// TIA Portal V15.1 export
// export: Created 2024-05-17T05:38:59.4838235Z, ExportSetting WithDefaults, DisplayName Totally Integrated Automation Portal, DisplayVersion V15.1 Update 5, DisplayName TIA Portal Openness, DisplayVersion V15.1 Update 5, DisplayName SINAMICS Startdrive Advanced, DisplayVersion V15.1, DisplayName G130, G150, S120, S150, SINAMICS MV, S210, DisplayVersion V15.1, DisplayName G110M, G120, G120C, G120D, G120P, DisplayVersion V15.1, DisplayName STEP 7 Professional, DisplayVersion V15.1 Update 5, DisplayName STEP 7 Safety, DisplayVersion V15.1, DisplayName WinCC Professional, DisplayVersion V15.1 Update 5, DisplayName SIMATIC Visualization Architect, DisplayVersion V15.1
FUNCTION "DiagPLCOverview" : Void   // FC251, FBD
TITLE = DiagPLCOverview
{ S7_Optimized_Access := 'FALSE' }
AUTHOR : VCC
NAME : LocFunc
VERSION : 0.1
// stored: AutoNumber false, IsIECCheckEnabled false, SetENOAutomatically False, UDAEnableTagReadback false
   VAR_OUTPUT
      O_AlarmA : Bool;   // Alarm A
      O_AlarmB : Bool;   // Alarm B
      O_AlarmC : Bool;   // Alarm C
      O_AlarmD : Bool;   // Alarm D
      O_AlarmABCondition : Bool;   // Alarms resetable
      H_IAnim : Word;   // Icon Animation
   END_VAR
   VAR_TEMP   // added for the SCL form of the ladder/FBD networks
      _w1 : Bool;
      _w2 : Bool;
   END_VAR
BEGIN

REGION Network 1: **** 1 - Inputs **** HMI Cmd
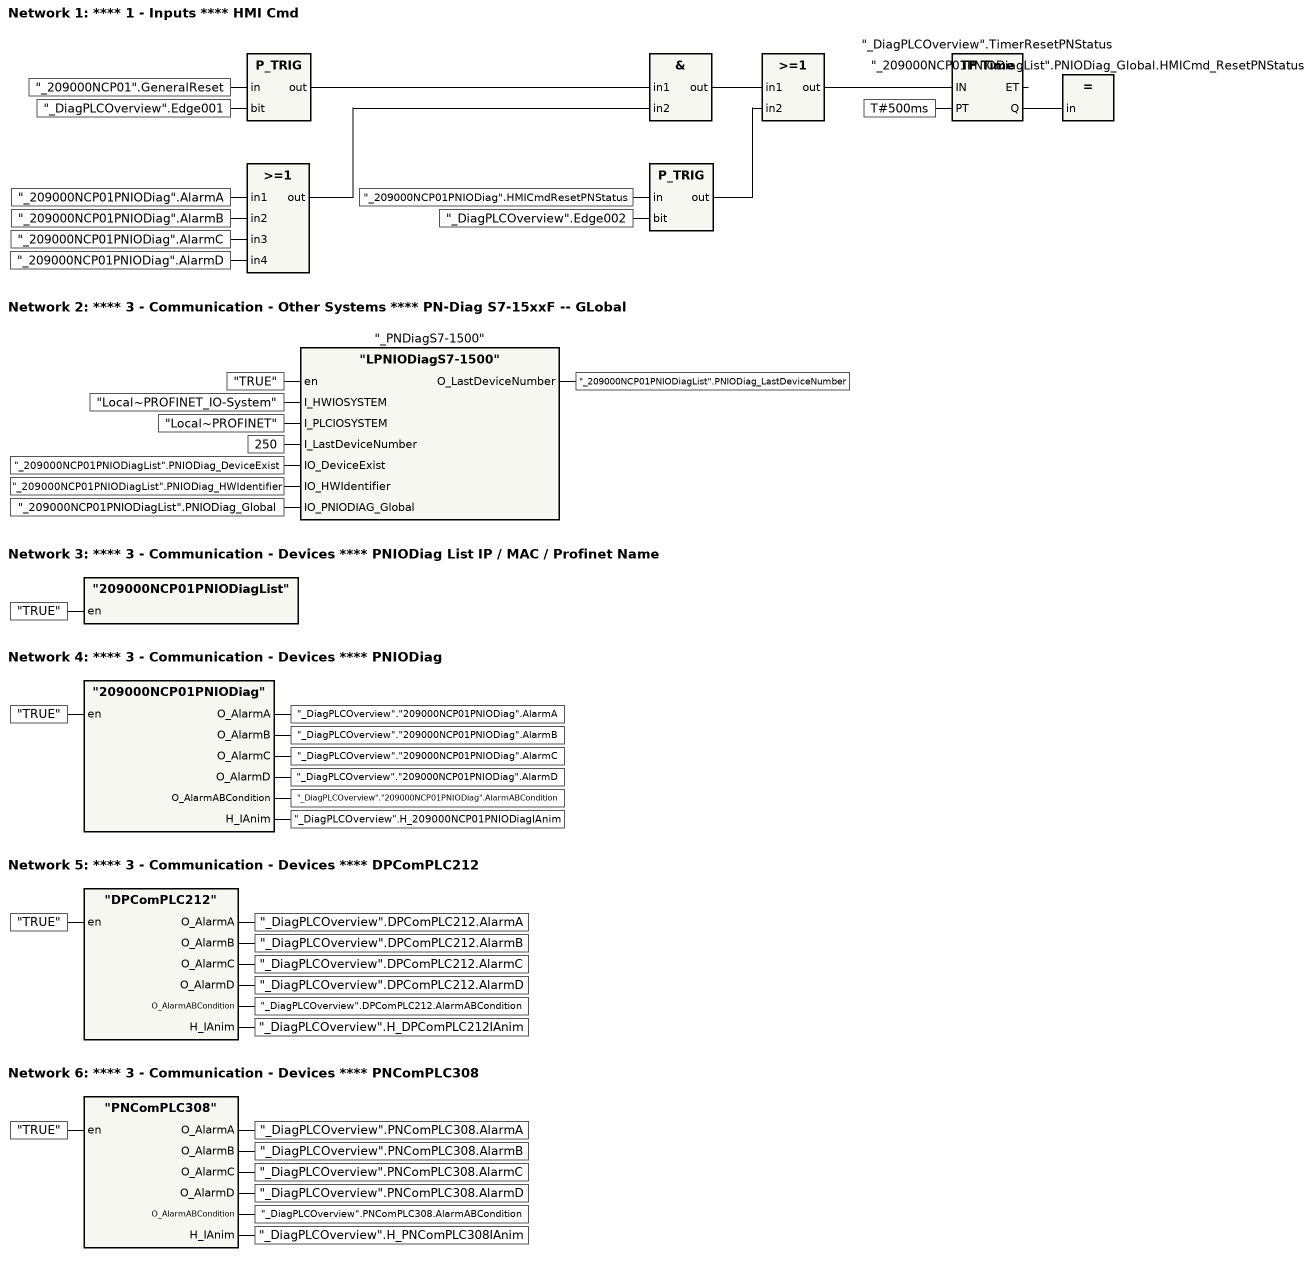
   #_w1 := "_209000NCP01".GeneralReset AND NOT "_DiagPLCOverview".Edge001;   // rising edge
   "_DiagPLCOverview".Edge001 := "_209000NCP01".GeneralReset;
   #_w2 := "_209000NCP01PNIODiag".HMICmdResetPNStatus AND NOT "_DiagPLCOverview".Edge002;   // rising edge
   "_DiagPLCOverview".Edge002 := "_209000NCP01PNIODiag".HMICmdResetPNStatus;
   "_DiagPLCOverview".TimerResetPNStatus.TP(IN := (#_w1 AND ("_209000NCP01PNIODiag".AlarmA OR "_209000NCP01PNIODiag".AlarmB OR "_209000NCP01PNIODiag".AlarmC OR "_209000NCP01PNIODiag".AlarmD)) OR #_w2,
                           PT := T#500ms);
   "_209000NCP01PNIODiagList".PNIODiag_Global.HMICmd_ResetPNStatus := "_DiagPLCOverview".TimerResetPNStatus.Q;
END_REGION

REGION Network 2: **** 3 - Communication - Other Systems **** PN-Diag S7-15xxF -- GLobal
   // PN-Diag S7-15xxF
   IF "TRUE" THEN
       "_PNDiagS7-1500"(I_HWIOSYSTEM := "Local~PROFINET_IO-System",   // "LPNIODiagS7-1500"
                        I_PLCIOSYSTEM := "Local~PROFINET",
                        I_LastDeviceNumber := 250,
                        IO_DeviceExist := "_209000NCP01PNIODiagList".PNIODiag_DeviceExist,
                        IO_HWIdentifier := "_209000NCP01PNIODiagList".PNIODiag_HWIdentifier,
                        IO_PNIODIAG_Global := "_209000NCP01PNIODiagList".PNIODiag_Global,
                        O_LastDeviceNumber => "_209000NCP01PNIODiagList".PNIODiag_LastDeviceNumber);
   END_IF;
END_REGION

REGION Network 3: **** 3 - Communication - Devices **** PNIODiag List IP / MAC / Profinet Name
   IF "TRUE" THEN "209000NCP01PNIODiagList"(); END_IF;
END_REGION

REGION Network 4: **** 3 - Communication - Devices **** PNIODiag
   IF "TRUE" THEN
       "209000NCP01PNIODiag"(O_AlarmA => "_DiagPLCOverview"."209000NCP01PNIODiag".AlarmA,
                             O_AlarmB => "_DiagPLCOverview"."209000NCP01PNIODiag".AlarmB,
                             O_AlarmC => "_DiagPLCOverview"."209000NCP01PNIODiag".AlarmC,
                             O_AlarmD => "_DiagPLCOverview"."209000NCP01PNIODiag".AlarmD,
                             O_AlarmABCondition => "_DiagPLCOverview"."209000NCP01PNIODiag".AlarmABCondition,
                             H_IAnim => "_DiagPLCOverview".H_209000NCP01PNIODiagIAnim);
   END_IF;
END_REGION

REGION Network 5: **** 3 - Communication - Devices **** DPComPLC212
   // DP/DP coupler communication
   IF "TRUE" THEN
       "DPComPLC212"(O_AlarmA => "_DiagPLCOverview".DPComPLC212.AlarmA,
                     O_AlarmB => "_DiagPLCOverview".DPComPLC212.AlarmB,
                     O_AlarmC => "_DiagPLCOverview".DPComPLC212.AlarmC,
                     O_AlarmD => "_DiagPLCOverview".DPComPLC212.AlarmD,
                     O_AlarmABCondition => "_DiagPLCOverview".DPComPLC212.AlarmABCondition,
                     H_IAnim => "_DiagPLCOverview".H_DPComPLC212IAnim);
   END_IF;
END_REGION

REGION Network 6: **** 3 - Communication - Devices **** PNComPLC308
   // PN/PN coupler communication
   IF "TRUE" THEN
       "PNComPLC308"(O_AlarmA => "_DiagPLCOverview".PNComPLC308.AlarmA,
                     O_AlarmB => "_DiagPLCOverview".PNComPLC308.AlarmB,
                     O_AlarmC => "_DiagPLCOverview".PNComPLC308.AlarmC,
                     O_AlarmD => "_DiagPLCOverview".PNComPLC308.AlarmD,
                     O_AlarmABCondition => "_DiagPLCOverview".PNComPLC308.AlarmABCondition,
                     H_IAnim => "_DiagPLCOverview".H_PNComPLC308IAnim);
   END_IF;
END_REGION

REGION Network 7: **** 3 - Communication - Devices **** VD Com
   // Virtual Device communication
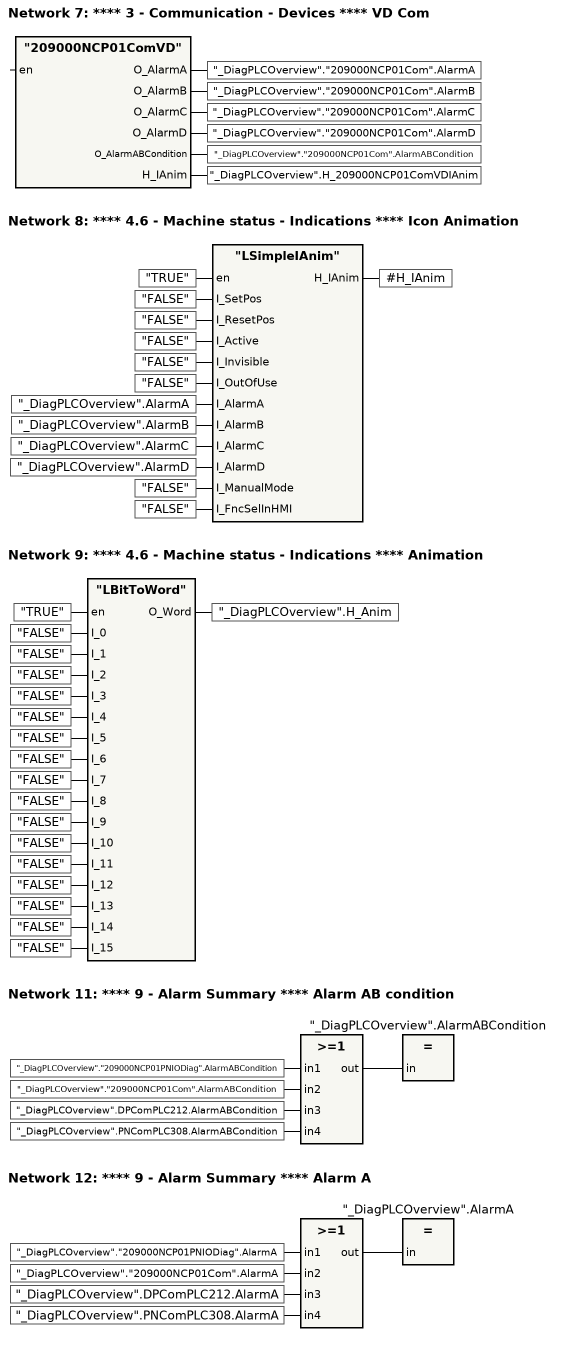
   "209000NCP01ComVD"(O_AlarmA => "_DiagPLCOverview"."209000NCP01Com".AlarmA,
                      O_AlarmB => "_DiagPLCOverview"."209000NCP01Com".AlarmB,
                      O_AlarmC => "_DiagPLCOverview"."209000NCP01Com".AlarmC,
                      O_AlarmD => "_DiagPLCOverview"."209000NCP01Com".AlarmD,
                      O_AlarmABCondition => "_DiagPLCOverview"."209000NCP01Com".AlarmABCondition,
                      H_IAnim => "_DiagPLCOverview".H_209000NCP01ComVDIAnim);
END_REGION

REGION Network 8: **** 4.6 - Machine status - Indications **** Icon Animation
   // Icon Animation for HMI
   IF "TRUE" THEN
       "LSimpleIAnim"(I_SetPos := "FALSE",
                      I_ResetPos := "FALSE",
                      I_Active := "FALSE",
                      I_Invisible := "FALSE",
                      I_OutOfUse := "FALSE",
                      I_AlarmA := "_DiagPLCOverview".AlarmA,
                      I_AlarmB := "_DiagPLCOverview".AlarmB,
                      I_AlarmC := "_DiagPLCOverview".AlarmC,
                      I_AlarmD := "_DiagPLCOverview".AlarmD,
                      I_ManualMode := "FALSE",
                      I_FncSelInHMI := "FALSE",
                      H_IAnim => #H_IAnim);
   END_IF;
END_REGION

REGION Network 9: **** 4.6 - Machine status - Indications **** Animation
   // Animation
   IF "TRUE" THEN
       "LBitToWord"(I_0 := "FALSE",
                    I_1 := "FALSE",
                    I_2 := "FALSE",
                    I_3 := "FALSE",
                    I_4 := "FALSE",
                    I_5 := "FALSE",
                    I_6 := "FALSE",
                    I_7 := "FALSE",
                    I_8 := "FALSE",
                    I_9 := "FALSE",
                    I_10 := "FALSE",
                    I_11 := "FALSE",
                    I_12 := "FALSE",
                    I_13 := "FALSE",
                    I_14 := "FALSE",
                    I_15 := "FALSE",
                    O_Word => "_DiagPLCOverview".H_Anim);
   END_IF;
END_REGION

NETWORK
TITLE = **** 4.6 - Machine Status - Indications **** Animation DB number
// DB number
      OPN   "_DiagPLCOverview";
      L     DBNO;
      T     "_DiagPLCOverview".H_DBnr;

REGION Network 11: **** 9 - Alarm Summary **** Alarm AB condition
   // Alarm AB condition
   "_DiagPLCOverview".AlarmABCondition := "_DiagPLCOverview"."209000NCP01PNIODiag".AlarmABCondition OR "_DiagPLCOverview"."209000NCP01Com".AlarmABCondition OR "_DiagPLCOverview".DPComPLC212.AlarmABCondition OR "_DiagPLCOverview".PNComPLC308.AlarmABCondition;
END_REGION

REGION Network 12: **** 9 - Alarm Summary **** Alarm A
   // Summary of alarms A
   "_DiagPLCOverview".AlarmA := "_DiagPLCOverview"."209000NCP01PNIODiag".AlarmA OR "_DiagPLCOverview"."209000NCP01Com".AlarmA OR "_DiagPLCOverview".DPComPLC212.AlarmA OR "_DiagPLCOverview".PNComPLC308.AlarmA;
END_REGION

REGION Network 13: **** 9 - Alarm Summary **** Alarm B
   // Summary of alarms B
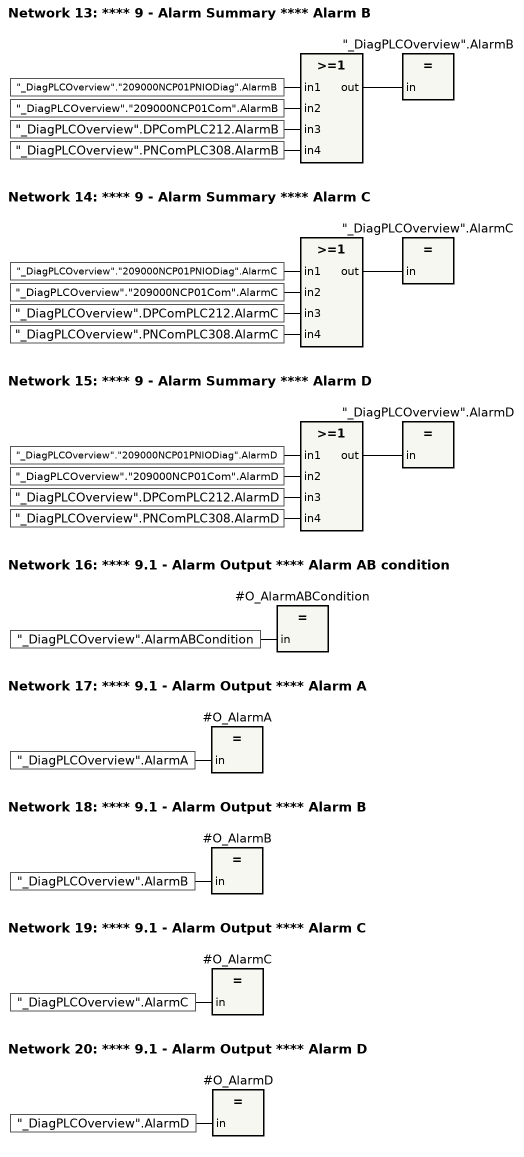
   "_DiagPLCOverview".AlarmB := "_DiagPLCOverview"."209000NCP01PNIODiag".AlarmB OR "_DiagPLCOverview"."209000NCP01Com".AlarmB OR "_DiagPLCOverview".DPComPLC212.AlarmB OR "_DiagPLCOverview".PNComPLC308.AlarmB;
END_REGION

REGION Network 14: **** 9 - Alarm Summary **** Alarm C
   // Summary of alarms C
   "_DiagPLCOverview".AlarmC := "_DiagPLCOverview"."209000NCP01PNIODiag".AlarmC OR "_DiagPLCOverview"."209000NCP01Com".AlarmC OR "_DiagPLCOverview".DPComPLC212.AlarmC OR "_DiagPLCOverview".PNComPLC308.AlarmC;
END_REGION

REGION Network 15: **** 9 - Alarm Summary **** Alarm D
   // Summary of alarms D
   "_DiagPLCOverview".AlarmD := "_DiagPLCOverview"."209000NCP01PNIODiag".AlarmD OR "_DiagPLCOverview"."209000NCP01Com".AlarmD OR "_DiagPLCOverview".DPComPLC212.AlarmD OR "_DiagPLCOverview".PNComPLC308.AlarmD;
END_REGION

REGION Network 16: **** 9.1 - Alarm Output **** Alarm AB condition
   // Alarm AB condition
   #O_AlarmABCondition := "_DiagPLCOverview".AlarmABCondition;
END_REGION

REGION Network 17: **** 9.1 - Alarm Output **** Alarm A
   // Summary of alarms A
   #O_AlarmA := "_DiagPLCOverview".AlarmA;
END_REGION

REGION Network 18: **** 9.1 - Alarm Output **** Alarm B
   // Summary of alarms B
   #O_AlarmB := "_DiagPLCOverview".AlarmB;
END_REGION

REGION Network 19: **** 9.1 - Alarm Output **** Alarm C
   // Summary of alarms C
   #O_AlarmC := "_DiagPLCOverview".AlarmC;
END_REGION

REGION Network 20: **** 9.1 - Alarm Output **** Alarm D
   // Summary of alarms D
   #O_AlarmD := "_DiagPLCOverview".AlarmD;
END_REGION

REGION Network 21: **** 9.2 - Alarm DWord**** Alarm To DWord
   // Alarm Word
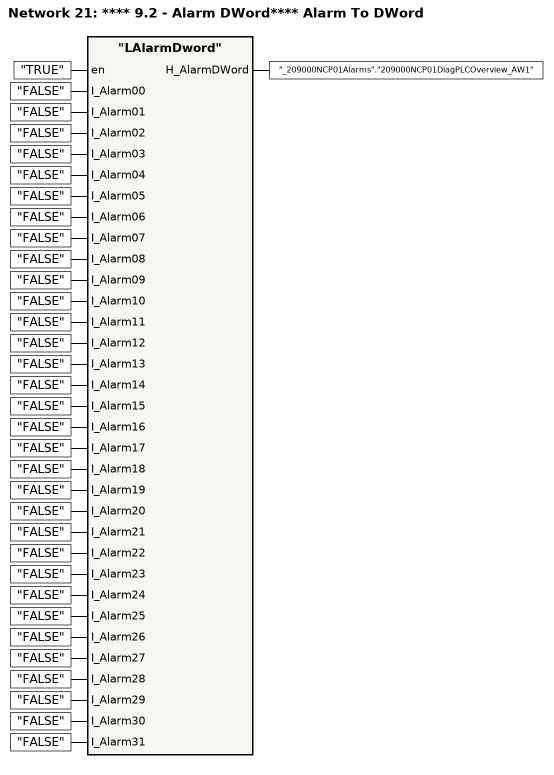
   IF "TRUE" THEN
       "LAlarmDword"(I_Alarm00 := "FALSE",
                     I_Alarm01 := "FALSE",
                     I_Alarm02 := "FALSE",
                     I_Alarm03 := "FALSE",
                     I_Alarm04 := "FALSE",
                     I_Alarm05 := "FALSE",
                     I_Alarm06 := "FALSE",
                     I_Alarm07 := "FALSE",
                     I_Alarm08 := "FALSE",
                     I_Alarm09 := "FALSE",
                     I_Alarm10 := "FALSE",
                     I_Alarm11 := "FALSE",
                     I_Alarm12 := "FALSE",
                     I_Alarm13 := "FALSE",
                     I_Alarm14 := "FALSE",
                     I_Alarm15 := "FALSE",
                     I_Alarm16 := "FALSE",
                     I_Alarm17 := "FALSE",
                     I_Alarm18 := "FALSE",
                     I_Alarm19 := "FALSE",
                     I_Alarm20 := "FALSE",
                     I_Alarm21 := "FALSE",
                     I_Alarm22 := "FALSE",
                     I_Alarm23 := "FALSE",
                     I_Alarm24 := "FALSE",
                     I_Alarm25 := "FALSE",
                     I_Alarm26 := "FALSE",
                     I_Alarm27 := "FALSE",
                     I_Alarm28 := "FALSE",
                     I_Alarm29 := "FALSE",
                     I_Alarm30 := "FALSE",
                     I_Alarm31 := "FALSE",
                     H_AlarmDWord => "_209000NCP01Alarms"."209000NCP01DiagPLCOverview_AW1");
   END_IF;
END_REGION
END_FUNCTION
